Universal Robots PolyScope program: SocketTest.urp

Program SocketTest (installation=default directory=/home/ur/ursim-current/programs createdIn=3.2.18654.0 lastSavedIn=3.11.0.82155 robotSerialNumber=20183099999)
Calibrated DH parameters: a=[0, -0.612, -0.5723, 0, 0, 0]; d=[0.1273, 0, 0, 0.163941, 0.1157, 0.0922]; alpha=[1.570796, 0, 0, 1.570796, -1.570796, 0]; deltaTheta=[0, 0, 0, 0, 0, 0]
BeforeStart
  Script file /home/ur/ursim-current/programs/JointFunction.script
    | global angles=[0,0,0,0,0,0]
    | global angles_send=""
    | 
    | sockon=socket_open("192.168.102.1",5000,"sock1")
    | def getjointAngles():
    | 	angles=get_actual_joint_positions()
    |                   angles_send=str_cat(angles[0],";")
    |  	angles_send=str_cat(angles_send,angles[1])
    | 	angles_send=str_cat(angles_send,";")
    | 	angles_send=str_cat(angles_send,angles[2])
    | 	angles_send=str_cat(angles_send,";")
    | 	angles_send=str_cat(angles_send,angles[3])
    | 	angles_send=str_cat(angles_send,";")
    | 	angles_send=str_cat(angles_send,angles[4])
    | 	angles_send=str_cat(angles_send,";")
    | 	angles_send=str_cat(angles_send,angles[5])
    | 	sockon= socket_send_line(angles_send)
    | 
    | 
    | end
Robot Program (runOnlyOnce=false)
  MoveJ speed 60 deg/s, acceleration 80 deg/s^2 (useActiveTCP=false)
    Waypoint Waypoint_1: TCP in base x=611.978 y=-161.7 z=230.789 mm, rx=2.2546 ry=-2.1864 rz=-0.0556 rad; joints [0, -98.956, -126.223, -46.295, 91.393, -1.776] deg
    Waypoint Waypoint_2: TCP in base x=161.7 y=611.978 z=230.789 mm, rx=3.1157 ry=0.0478 rz=-0.0385 rad; joints [90, -98.956, -126.223, -46.295, 91.393, -1.776] deg
Thread Thread_1 (runOnlyOnce=false)
  Loop While (checkContinuously=true) expression=sockon≟ True
    Script: getjointAngles()
    Wait Sleep waitTime=0.05
  If sockon≟ False
    Script: socket_close("sock1")
    Script: sockon=socket_open("192.168.102.1",5000)
    Wait Sleep waitTime=0.01
